// TODO rename + your commands
{attribute 'qualified_only'}
TYPE E_TemplateCommand : (NONE := 0, DO_A := 1, DO_B := 2) DINT;
END_TYPE

(* stored: Version 1.1.0.1, ProductVersion 3.1.4024.12
   DUT E_TemplateCommand: Id {430177f0-5378-4a81-9dbf-9c1074728d73} *)
